// TIA Portal V20 export
DATA_BLOCK "EM_MonitorData"   // DB373
// stored: MemoryReserve 100, Namespace Unit1
   VAR
      EM00 : Struct
         Spare_bit : Bool;
      END_STRUCT;
      EM01 : Struct
         Spare_bit : Bool;
      END_STRUCT;
      EM02 : Struct
         jrOutPnPLeft : Struct
            WorkDonw : Struct
               stack1LoadJob2 : Bool;
               stack2LoadJob3 : Bool;
               unloadJob4 : Bool;
            END_STRUCT;
         END_STRUCT;
         jrOutPnPRight : Struct
            WorkDone : Struct
               loadJob2 : Bool;
               unloadJob3 : Bool;
            END_STRUCT;
         END_STRUCT;
      END_STRUCT;
      EM03 : Struct
         topTapeLoading : Struct
            WorkDonw : Struct
               chargeJob2 : Bool;
            END_STRUCT;
         END_STRUCT;
         topTapeAttachment : Struct
            WorkDone : Struct
               tapeGetJob2 : Bool;
               tape1PutJob3 : Bool;
               tape2PutJob4 : Bool;
               tapeIdleJob5 : Bool;
            END_STRUCT;
         END_STRUCT;
         topTapeFixStage : Struct
            WorkDone : Struct
               loadJob2 : Bool;
               taping1Job3 : Bool;
               taping2Job4 : Bool;
               unloadJob5 : Bool;
            END_STRUCT;
         END_STRUCT;
      END_STRUCT;
      EM04 : Struct
         sideTapeLoading : Struct
            WorkDone : Bool;
         END_STRUCT;
         sideTapeAttachment : Struct
            WorkDone : Struct
               rightTapeGetJob2 : Bool;
               leftTapeGetJob3 : Bool;
               tape1PutJob4 : Bool;
               tape2PutJob5 : Bool;
               tape3PutJob6 : Bool;
               tape4PutJob7 : Bool;
               TapeIdleJob8 : Bool;
            END_STRUCT;
         END_STRUCT;
         sideTapeFixStage : Struct
            WorkDone : Struct
               loadJob2 : Bool;
               taping1Job3 : Bool;
               taping2Job4 : Bool;
               taping3Job5 : Bool;
               taping4Job6 : Bool;
               unloadJob7 : Bool;
            END_STRUCT;
         END_STRUCT;
      END_STRUCT;
      EM05 : Struct
         transferPnPLeft : Struct
            WorkDone : Struct
               sideTapeLoadJob2_A : Bool;
               hotPressLeftUnloadJob3_A : Bool;
               hotPressLeftLoadJob4_A : Bool;
               sideTapeLoadJob5_B : Bool;
               hotPressRightUnloadJob6_B : Bool;
               hotPressRightLoadJob7_B : Bool;
               hipotThicknessUnloadJob9 : Bool;
            END_STRUCT;
         END_STRUCT;
         transferPnPRight : Struct
            WorkDone : Struct
               hipotThicknessLoadJob2 : Bool;
               visionUnloadJob3 : Bool;
               visionLoadJob4 : Bool;
               laserMarkUnloadJob5 : Bool;
               laserMarkLoadJob6 : Bool;
               weightCheckUnloadJob9 : Bool;
            END_STRUCT;
         END_STRUCT;
         GRnR_TransferPnP : Struct
            WorkDone : Struct
               transferPnPLeft : Bool;
               transferPnPRight : Bool;
            END_STRUCT;
         END_STRUCT;
      END_STRUCT;
      EM06 : Struct
         WorkDone : Struct
            LoadJob2 : Bool;
            InspectionJob3 : Bool;
            UnloadJob4 : Bool;
         END_STRUCT;
      END_STRUCT;
      EM07 : Struct
         WorkDone : Struct
            LoadJob2 : Bool;
            InspectionJob3 : Bool;
            UnloadJob4 : Bool;
         END_STRUCT;
      END_STRUCT;
      EM08 : Struct
         WorkDone : Struct
            LoadJob2 : Bool;
            InspectionJob3 : Bool;
            UnloadJob4 : Bool;
         END_STRUCT;
      END_STRUCT;
      EM09 : Struct
         WorkDone : Struct
            LoadJob2 : Bool;
            InspectionJob3 : Bool;
            UnloadJob4 : Bool;
         END_STRUCT;
      END_STRUCT;
      EM10 : Struct
         WorkDone : Struct
            LoadJob2 : Bool;
            InspectionJob3 : Bool;
            UnloadJob4 : Bool;
         END_STRUCT;
      END_STRUCT;
      EM11 : Struct
         WorkDone : Struct
            LoadJob2 : Bool;
            InspectionJob3 : Bool;
            UnloadJob4 : Bool;
         END_STRUCT;
      END_STRUCT;
      EM12 : Struct
         Spare_bit : Bool;
      END_STRUCT;
      EM13 : Struct
         Spare_bit : Bool;
      END_STRUCT;
   END_VAR
BEGIN
END_DATA_BLOCK
